FUNCTION_BLOCK EmergencyInit2 (* CAT Function Block Type *)
  (* Standard: 61499-2 *)
  (* Version 0.0, 7/15/2026, Schneider Electric, template *)
  PACKAGE SE.Nereda;
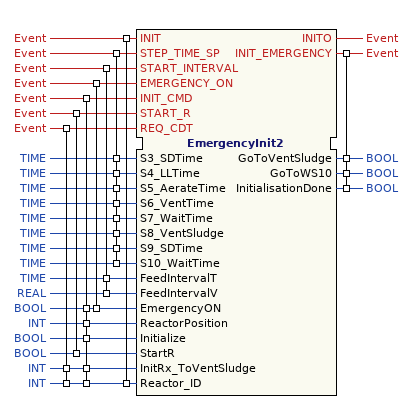
  EVENT_INPUT
    INIT WITH Reactor_ID;
    STEP_TIME_SP WITH S3_SDTime, S4_LLTime, S5_AerateTime, S6_VentTime, S7_WaitTime, S8_VentSludge, S9_SDTime, S10_WaitTime;
    START_INTERVAL WITH FeedIntervalT, FeedIntervalV;
    EMERGENCY_ON WITH EmergencyON;
    INIT_CMD WITH EmergencyON, ReactorPosition, Initialize, InitRx_ToVentSludge, Reactor_ID;
    START_R WITH StartR;
    REQ_CDT WITH InitRx_ToVentSludge, Reactor_ID;
  END_EVENT
  EVENT_OUTPUT
    INITO;
    INIT_EMERGENCY WITH GoToVentSludge, GoToWS10, InitialisationDone;
  END_EVENT
  VAR_INPUT
    S3_SDTime : TIME;
    S4_LLTime : TIME;
    S5_AerateTime : TIME;
    S6_VentTime : TIME;
    S7_WaitTime : TIME;
    S8_VentSludge : TIME;
    S9_SDTime : TIME;
    S10_WaitTime : TIME;
    FeedIntervalT : TIME;
    FeedIntervalV : REAL;
    EmergencyON : BOOL;
    ReactorPosition : INT;
    Initialize : BOOL;
    StartR : BOOL;
    InitRx_ToVentSludge : INT;
    Reactor_ID : INT;
  END_VAR
  VAR_OUTPUT
    GoToVentSludge : BOOL;
    GoToWS10 : BOOL;
    InitialisationDone : BOOL;
  END_VAR
  (* 01 - FUNCTIONNAL INPUT INTERFACE *)
  (* 00 - INITIALIZATION *)
  (* 05 - LOGIC *)
  (* 06 - HMI INTERFACE *)
  (* 03 - FIELD INTERFACE *)
  (* 02 - FUNCTIONNAL OUTPUT INTERFACE *)
  (* Logic *)
  (* 04 - CHILDREN *)
  (* 4A - TYPICALS *)
  FBS
    IThis : EmergencyInit2_HMI(QI := TRUE);
    EnoughTime : StepRestOfTimeCalc2;
    Time2Real : TIME2REAL_8;
    DecideInit : EmergencyDecideInit2;
    msToMin : DIVIDE(pin_02E479D09E2C7EA2 := 1000);
    Init : E_PERMIT;
  END_FBS
  EVENT_CONNECTIONS
    INIT TO IThis.93BB138255CAD99E;
    IThis.6860A233C9096CA6 TO INITO;
    START_INTERVAL TO Time2Real.9954577AA24F9DD6;
    STEP_TIME_SP TO Time2Real.9954577AA24F9DD6;
    Time2Real.79B40746AB555956 TO msToMin.0FDF8A587C3CA146;
    EnoughTime.50D90A5AAF562FFD TO DecideInit.A265894F67E5210F;
    DecideInit.BCEA9B57A1625B8E TO INIT_EMERGENCY;
    Init.EO TO DecideInit.CB5BC2F1A1AE16A3;
    EMERGENCY_ON TO Time2Real.9954577AA24F9DD6;
    msToMin.6D05A744943B688E TO EnoughTime.DE3F91074AB90905;
    INIT_CMD TO Init.EI;
    START_R TO DecideInit.BB0EC835D9E6E7EC;
    REQ_CDT TO DecideInit.EBD053A98A1A70A5;
    EMERGENCY_ON TO DecideInit.EBD053A98A1A70A5;
  END_CONNECTIONS
  DATA_CONNECTIONS
    FeedIntervalV TO msToMin.8EF5C40F2FEA5451;
    Time2Real.8AC404843F53B283 TO EnoughTime.F22EA5F248A50CC4;
    Time2Real.FADDF116EEE78DD8 TO EnoughTime.BA6E402D256389C3;
    Time2Real.F0AD27F053D1AF98 TO EnoughTime.99CDBF035F753575;
    Time2Real.B25DE754B5185002 TO EnoughTime.4007F4626DF49643;
    Time2Real.AAB73CAB4AE993B0 TO EnoughTime.40853A2DDC4FBA1A;
    Time2Real.4D1507586A17112D TO EnoughTime.31B01DC205FFD47B;
    S3_SDTime TO Time2Real.158B8AA7B31D2617;
    S4_LLTime TO Time2Real.00D88FA23835E0F1;
    S5_AerateTime TO Time2Real.E3DD408A3DDFE25F;
    S6_VentTime TO Time2Real.3F7EBA5693CD820C;
    S7_WaitTime TO Time2Real.DA4C33EA471E5B04;
    S8_VentSludge TO Time2Real.E244C798548C3E17;
    EnoughTime.E0E78CD8F23592D1 TO DecideInit.02AAB2707FF1365A;
    DecideInit.507EF3B39A4900A8 TO GoToVentSludge;
    DecideInit.D53B1E868844A93D TO GoToWS10;
    EmergencyON TO DecideInit.B4FF674B444ECDD1;
    ReactorPosition TO DecideInit.44B3F632AE826032;
    msToMin.E78A8A65D4120686 TO EnoughTime.A2F4F2631E28A856;
    Initialize TO Init.PERMIT;
    StartR TO DecideInit.D52D8FD10A41816B;
    DecideInit.26198284473355E5 TO InitialisationDone;
    InitRx_ToVentSludge TO DecideInit.E2AC83895D726999;
    Reactor_ID TO DecideInit.6F6BBDAF0E4B9539;
    S9_SDTime TO Time2Real.6CF2D7B11EFAFF1A;
    S10_WaitTime TO Time2Real.FC82385BB5F14083;
    Time2Real.B08BD2B776FAB925 TO EnoughTime.2AC8B971A669927E;
    Time2Real.C47B40E937652866 TO EnoughTime.3514E44EA39D1D5E;
  END_CONNECTIONS
END_FUNCTION_BLOCK
